Fanuc KAREL source: kc00034.KL

-- PROVISIONAL review KL for V940-1; original PC SHA256 3b09565439b2471c16e5822dbe00c9470edc5455cdea52ca0ecb735d4ddaf17b
-- Incomplete behavior may be omitted. Consult companion uncertainty JSON. Do not deploy.
PROGRAM KC00034
%NOLOCKGROUP
BEGIN
  -- V9_ZERO_TABLE_METADATA_HINT layout=0002_ascii; no indexed target words; source/name/runtime held
  -- UNRESOLVED_PC offsets 5-29; opcodes 27,22,22,2A,22,31
  -- UNRESOLVED_PC offsets 34-38; opcodes 7F
END KC00034
